// TIA Portal V18 export
FUNCTION "ST10_Main" : Void   // FC1050, LAD
{ S7_Optimized_Access := 'FALSE' }
VERSION : 0.1
// stored: AutoNumber false, IsIECCheckEnabled false, SetENOAutomatically false, UDAEnableTagReadback false
BEGIN

REGION Network 1
   // 系统功能组调用部分
   // 1.该部分用户可以自己根据系统的组成将需要的功能块调用写在该部分
   // 2.该部分禁止与系统功能无关的程序在此处调用
END_REGION

NETWORK
TITLE = XXXX=====Station Relation/工位相关 =====StartXXXXX / XXXX=====Station Relation/Station correlation =====StartXXXXX

REGION Network 3: input /输入
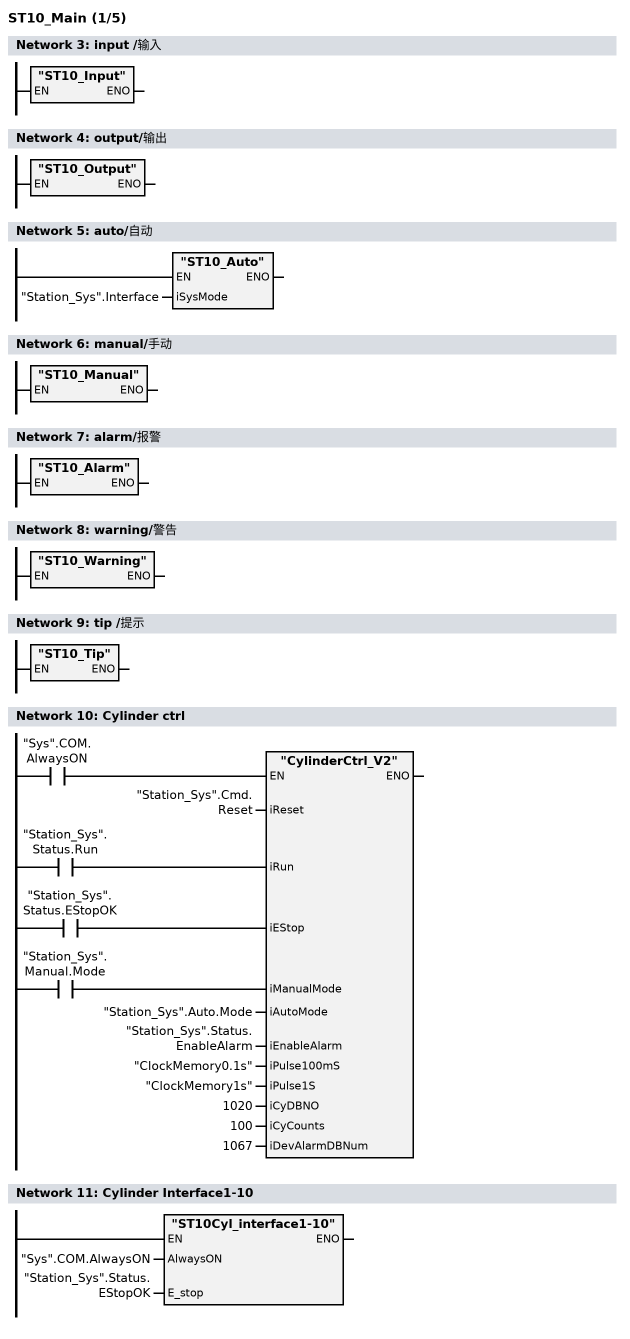
   RUNG wire#powerrail
      "ST10_Input"()
   END_RUNG
   // the same network as SCL:
   "ST10_Input"();
END_REGION

REGION Network 4: output/输出
   RUNG wire#powerrail
      "ST10_Output"()
   END_RUNG
   // the same network as SCL:
   "ST10_Output"();
END_REGION

REGION Network 5: auto/自动
   RUNG wire#powerrail
      "ST10_Auto"(iSysMode := "Station_Sys".Interface)
   END_RUNG
   // the same network as SCL:
   "ST10_Auto"(iSysMode := "Station_Sys".Interface);
END_REGION

REGION Network 6: manual/手动
   RUNG wire#powerrail
      "ST10_Manual"()
   END_RUNG
   // the same network as SCL:
   "ST10_Manual"();
END_REGION

REGION Network 7: alarm/报警
   RUNG wire#powerrail
      "ST10_Alarm"()
   END_RUNG
   // the same network as SCL:
   "ST10_Alarm"();
END_REGION

REGION Network 8: warning/警告
   RUNG wire#powerrail
      "ST10_Warning"()
   END_RUNG
   // the same network as SCL:
   "ST10_Warning"();
END_REGION

REGION Network 9: tip /提示
   RUNG wire#powerrail
      "ST10_Tip"()
   END_RUNG
   // the same network as SCL:
   "ST10_Tip"();
END_REGION

REGION Network 10: Cylinder ctrl
   RUNG wire#powerrail
      Contact( "Sys".COM.AlwaysON )
      "CylinderCtrl_V2"(iRun := wire#w1, iEStop := wire#w2, iManualMode := wire#w3, iReset := "Station_Sys".Cmd.Reset, iAutoMode := "Station_Sys".Auto.Mode, iEnableAlarm := "Station_Sys".Status.EnableAlarm, iPulse100mS := "ClockMemory0.1s", iPulse1S := "ClockMemory1s", iCyDBNO := 1020, iCyCounts := 100, iDevAlarmDBNum := 1067)
   END_RUNG
   RUNG wire#powerrail
      Contact( "Station_Sys".Status.Run )
   END_RUNG wire#w1
   RUNG wire#powerrail
      Contact( "Station_Sys".Status.EStopOK )
   END_RUNG wire#w2
   RUNG wire#powerrail
      Contact( "Station_Sys".Manual.Mode )
   END_RUNG wire#w3
   // the same network as SCL:
   IF "Sys".COM.AlwaysON THEN
       "CylinderCtrl_V2"(iReset := "Station_Sys".Cmd.Reset,
                         iRun := "Station_Sys".Status.Run,
                         iEStop := "Station_Sys".Status.EStopOK,
                         iManualMode := "Station_Sys".Manual.Mode,
                         iAutoMode := "Station_Sys".Auto.Mode,
                         iEnableAlarm := "Station_Sys".Status.EnableAlarm,
                         iPulse100mS := "ClockMemory0.1s",
                         iPulse1S := "ClockMemory1s",
                         iCyDBNO := 1020,
                         iCyCounts := 100,
                         iDevAlarmDBNum := 1067);
   END_IF;
END_REGION

REGION Network 11: Cylinder Interface1-10
   RUNG wire#powerrail
      "ST10Cyl_interface1-10"(AlwaysON := "Sys".COM.AlwaysON, E_stop := "Station_Sys".Status.EStopOK)
   END_RUNG
   // the same network as SCL:
   "ST10Cyl_interface1-10"(AlwaysON := "Sys".COM.AlwaysON, E_stop := "Station_Sys".Status.EStopOK);
END_REGION

REGION Network 12: Cylinder Interface11-20
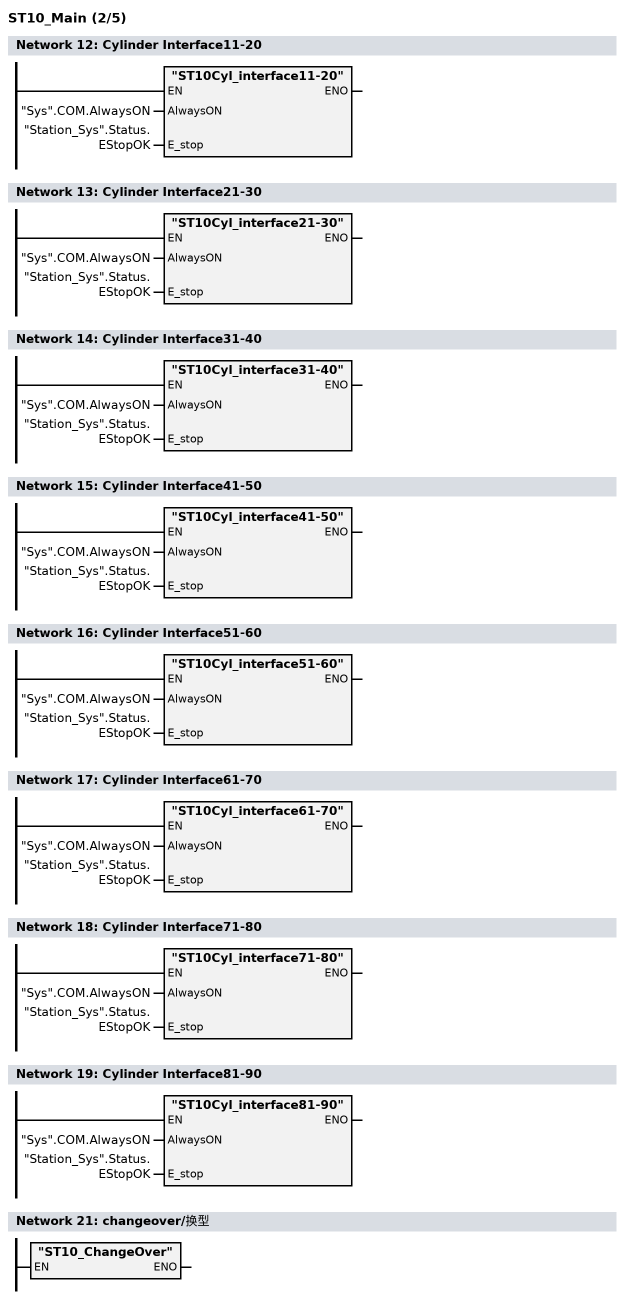
   RUNG wire#powerrail
      "ST10Cyl_interface11-20"(AlwaysON := "Sys".COM.AlwaysON, E_stop := "Station_Sys".Status.EStopOK)
   END_RUNG
   // the same network as SCL:
   "ST10Cyl_interface11-20"(AlwaysON := "Sys".COM.AlwaysON, E_stop := "Station_Sys".Status.EStopOK);
END_REGION

REGION Network 13: Cylinder Interface21-30
   RUNG wire#powerrail
      "ST10Cyl_interface21-30"(AlwaysON := "Sys".COM.AlwaysON, E_stop := "Station_Sys".Status.EStopOK)
   END_RUNG
   // the same network as SCL:
   "ST10Cyl_interface21-30"(AlwaysON := "Sys".COM.AlwaysON, E_stop := "Station_Sys".Status.EStopOK);
END_REGION

REGION Network 14: Cylinder Interface31-40
   RUNG wire#powerrail
      "ST10Cyl_interface31-40"(AlwaysON := "Sys".COM.AlwaysON, E_stop := "Station_Sys".Status.EStopOK)
   END_RUNG
   // the same network as SCL:
   "ST10Cyl_interface31-40"(AlwaysON := "Sys".COM.AlwaysON, E_stop := "Station_Sys".Status.EStopOK);
END_REGION

REGION Network 15: Cylinder Interface41-50
   RUNG wire#powerrail
      "ST10Cyl_interface41-50"(AlwaysON := "Sys".COM.AlwaysON, E_stop := "Station_Sys".Status.EStopOK)
   END_RUNG
   // the same network as SCL:
   "ST10Cyl_interface41-50"(AlwaysON := "Sys".COM.AlwaysON, E_stop := "Station_Sys".Status.EStopOK);
END_REGION

REGION Network 16: Cylinder Interface51-60
   RUNG wire#powerrail
      "ST10Cyl_interface51-60"(AlwaysON := "Sys".COM.AlwaysON, E_stop := "Station_Sys".Status.EStopOK)
   END_RUNG
   // the same network as SCL:
   "ST10Cyl_interface51-60"(AlwaysON := "Sys".COM.AlwaysON, E_stop := "Station_Sys".Status.EStopOK);
END_REGION

REGION Network 17: Cylinder Interface61-70
   RUNG wire#powerrail
      "ST10Cyl_interface61-70"(AlwaysON := "Sys".COM.AlwaysON, E_stop := "Station_Sys".Status.EStopOK)
   END_RUNG
   // the same network as SCL:
   "ST10Cyl_interface61-70"(AlwaysON := "Sys".COM.AlwaysON, E_stop := "Station_Sys".Status.EStopOK);
END_REGION

REGION Network 18: Cylinder Interface71-80
   RUNG wire#powerrail
      "ST10Cyl_interface71-80"(AlwaysON := "Sys".COM.AlwaysON, E_stop := "Station_Sys".Status.EStopOK)
   END_RUNG
   // the same network as SCL:
   "ST10Cyl_interface71-80"(AlwaysON := "Sys".COM.AlwaysON, E_stop := "Station_Sys".Status.EStopOK);
END_REGION

REGION Network 19: Cylinder Interface81-90
   RUNG wire#powerrail
      "ST10Cyl_interface81-90"(AlwaysON := "Sys".COM.AlwaysON, E_stop := "Station_Sys".Status.EStopOK)
   END_RUNG
   // the same network as SCL:
   "ST10Cyl_interface81-90"(AlwaysON := "Sys".COM.AlwaysON, E_stop := "Station_Sys".Status.EStopOK);
END_REGION

REGION Network 21: changeover/换型
   RUNG wire#powerrail
      "ST10_ChangeOver"()
   END_RUNG
   // the same network as SCL:
   "ST10_ChangeOver"();
END_REGION

REGION Network 22: Device
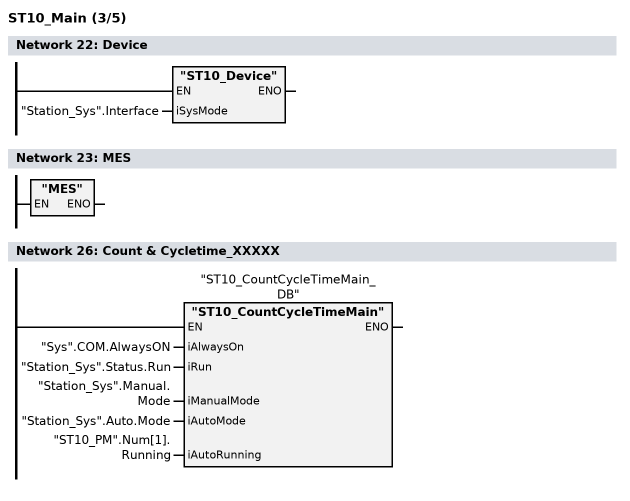
   RUNG wire#powerrail
      "ST10_Device"(iSysMode := "Station_Sys".Interface)
   END_RUNG
   // the same network as SCL:
   "ST10_Device"(iSysMode := "Station_Sys".Interface);
END_REGION

REGION Network 23: MES
   RUNG wire#powerrail
      "MES"()
   END_RUNG
   // the same network as SCL:
   "MES"();
END_REGION

REGION Network 24: =====System Function related information Section =====Start
END_REGION

NETWORK
TITLE = SystemFunction IO

REGION Network 26: Count & Cycletime_XXXXX
   RUNG wire#powerrail
      "ST10_CountCycleTimeMain_DB"(iAlwaysOn := "Sys".COM.AlwaysON, iRun := "Station_Sys".Status.Run, iManualMode := "Station_Sys".Manual.Mode, iAutoMode := "Station_Sys".Auto.Mode, iAutoRunning := "ST10_PM".Num[1].Running)
   END_RUNG
   // the same network as SCL:
   "ST10_CountCycleTimeMain_DB"(iAlwaysOn := "Sys".COM.AlwaysON,   // "ST10_CountCycleTimeMain"
                           iRun := "Station_Sys".Status.Run,
                           iManualMode := "Station_Sys".Manual.Mode,
                           iAutoMode := "Station_Sys".Auto.Mode,
                           iAutoRunning := "ST10_PM".Num[1].Running);
END_REGION

REGION Network 27: System mode
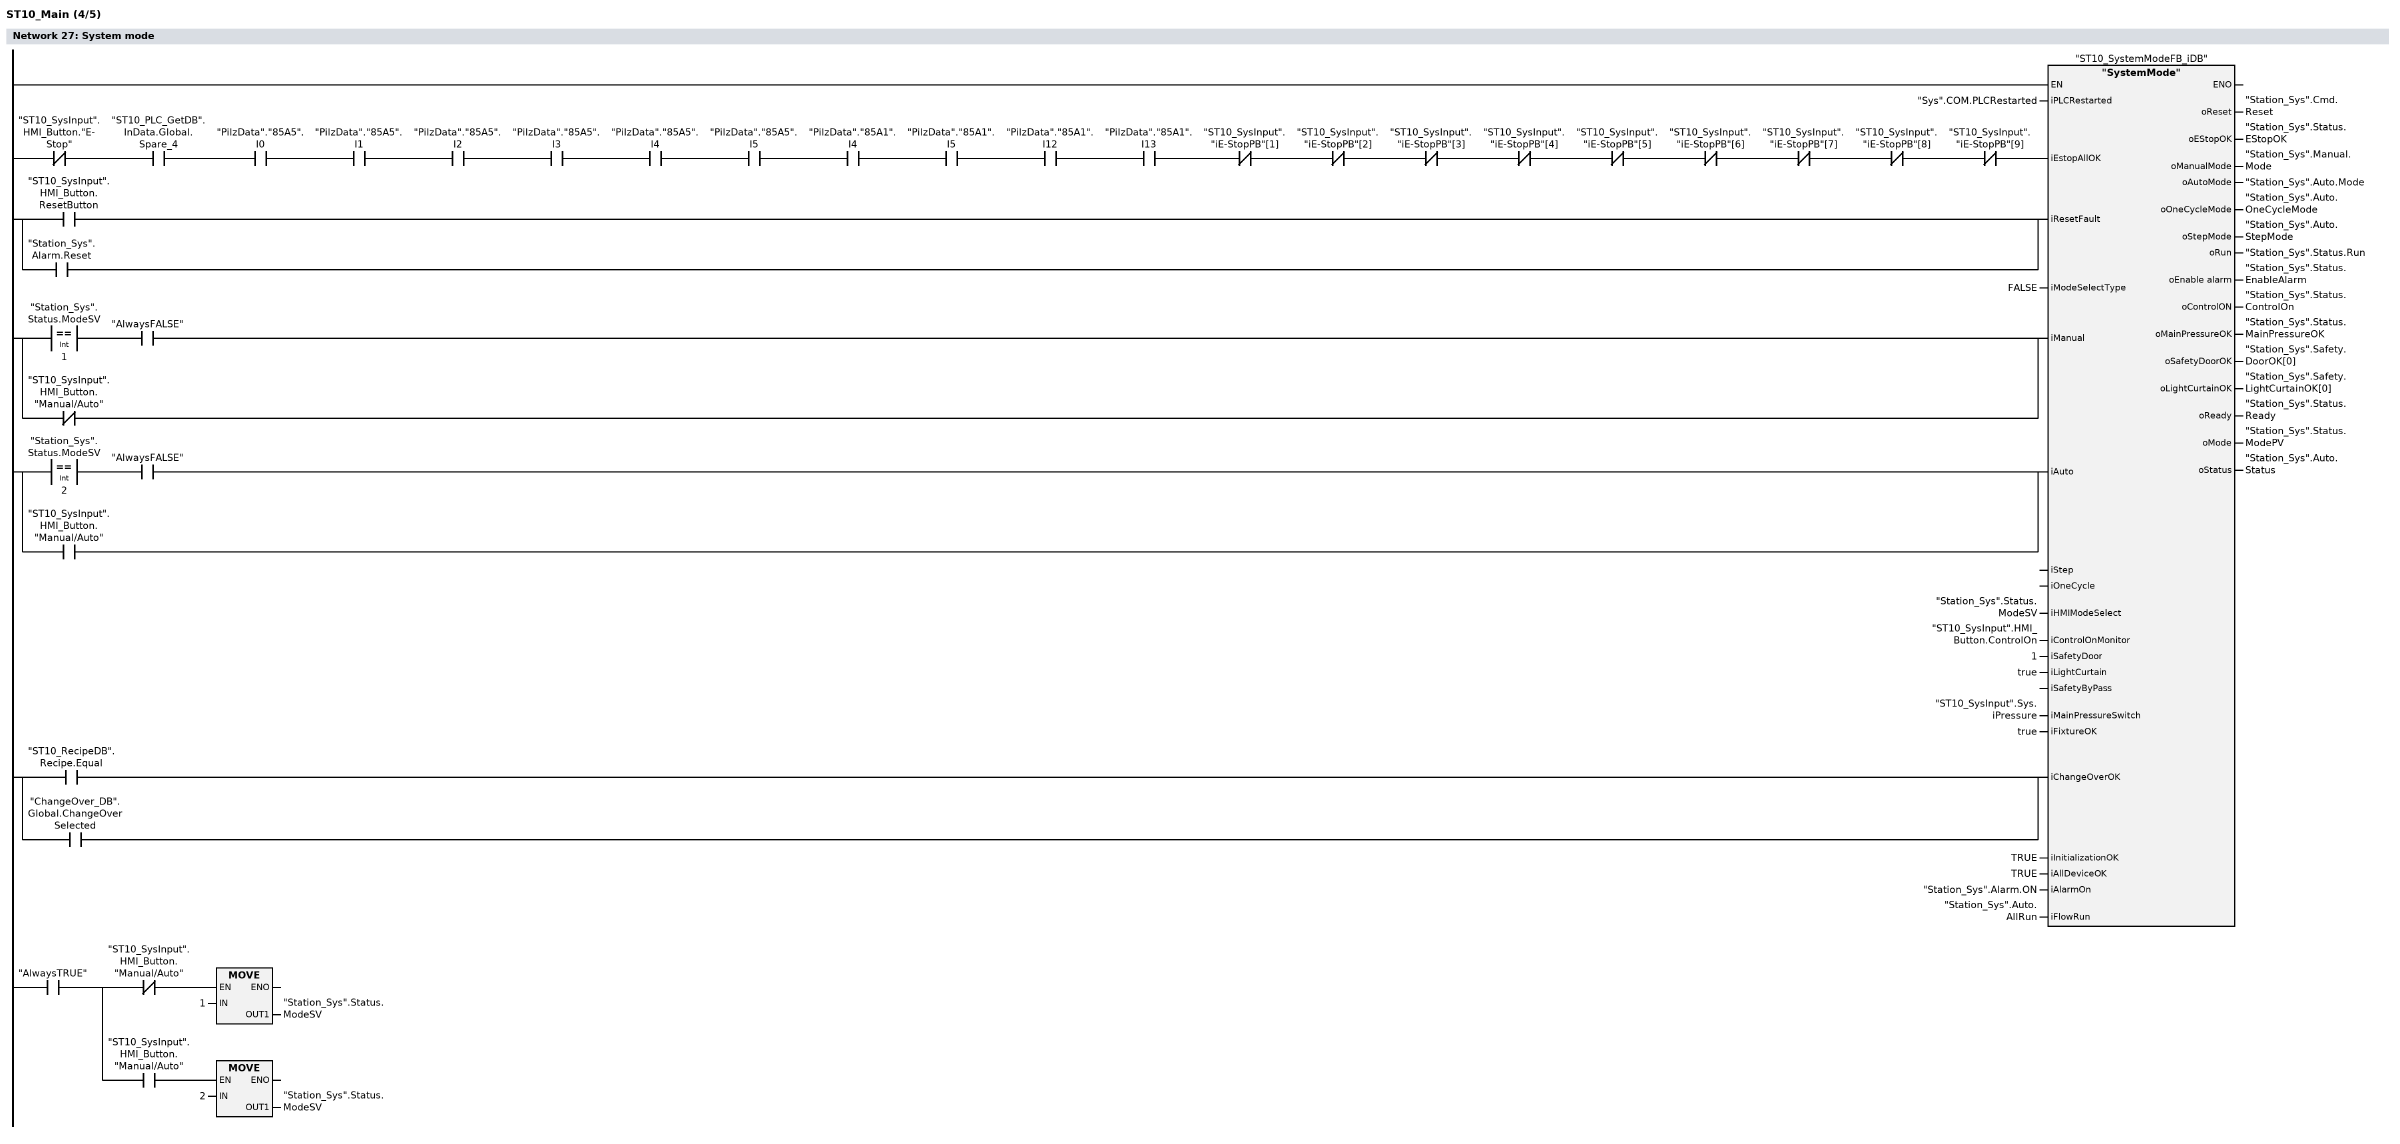
   RUNG wire#powerrail
      "ST10_SystemModeFB_iDB"(iEstopAllOK := wire#w1, iResetFault := wire#w2, iManual := wire#w3, iAuto := wire#w4, iChangeOverOK := wire#w5, iPLCRestarted := "Sys".COM.PLCRestarted, iModeSelectType := FALSE, iStep :=, iOneCycle :=, iHMIModeSelect := "Station_Sys".Status.ModeSV, iControlOnMonitor := "ST10_SysInput".HMI_Button.ControlOn, iSafetyDoor := 1, iLightCurtain := true, iSafetyByPass :=, iMainPressureSwitch := "ST10_SysInput".Sys.iPressure, iFixtureOK := true, iInitializationOK := TRUE, iAllDeviceOK := TRUE, iAlarmOn := "Station_Sys".Alarm.ON, iFlowRun := "Station_Sys".Auto.AllRun, oReset => "Station_Sys".Cmd.Reset, oEStopOK => "Station_Sys".Status.EStopOK, oManualMode => "Station_Sys".Manual.Mode, oAutoMode => "Station_Sys".Auto.Mode, oOneCycleMode => "Station_Sys".Auto.OneCycleMode, oStepMode => "Station_Sys".Auto.StepMode, oRun => "Station_Sys".Status.Run, "oEnable alarm" => "Station_Sys".Status.EnableAlarm, oControlON => "Station_Sys".Status.ControlOn, oMainPressureOK => "Station_Sys".Status.MainPressureOK, oSafetyDoorOK => "Station_Sys".Safety.DoorOK[0], oLightCurtainOK => "Station_Sys".Safety.LightCurtainOK[0], oReady => "Station_Sys".Status.Ready, oMode => "Station_Sys".Status.ModePV, oStatus => "Station_Sys".Auto.Status)
   END_RUNG
   RUNG wire#powerrail
      I_Contact( "ST10_SysInput".HMI_Button."E-Stop" )
      Contact( "ST10_PLC_GetDB".InData.Global.Spare_4 )
      Contact( "PilzData"."85A5".I0 )
      Contact( "PilzData"."85A5".I1 )
      Contact( "PilzData"."85A5".I2 )
      Contact( "PilzData"."85A5".I3 )
      Contact( "PilzData"."85A5".I4 )
      Contact( "PilzData"."85A5".I5 )
      Contact( "PilzData"."85A1".I4 )
      Contact( "PilzData"."85A1".I5 )
      Contact( "PilzData"."85A1".I12 )
      Contact( "PilzData"."85A1".I13 )
      I_Contact( "ST10_SysInput"."iE-StopPB"[1] )
      I_Contact( "ST10_SysInput"."iE-StopPB"[2] )
      I_Contact( "ST10_SysInput"."iE-StopPB"[3] )
      I_Contact( "ST10_SysInput"."iE-StopPB"[4] )
      I_Contact( "ST10_SysInput"."iE-StopPB"[5] )
      I_Contact( "ST10_SysInput"."iE-StopPB"[6] )
      I_Contact( "ST10_SysInput"."iE-StopPB"[7] )
      I_Contact( "ST10_SysInput"."iE-StopPB"[8] )
      I_Contact( "ST10_SysInput"."iE-StopPB"[9] )
   END_RUNG wire#w1
   RUNG wire#powerrail
      Contact( "ST10_SysInput".HMI_Button.ResetButton )
   END_RUNG wire#w2
   RUNG wire#powerrail
      Contact( "Station_Sys".Alarm.Reset )
   END_RUNG wire#w2
   RUNG wire#powerrail
      { S7_Templates := "SrcType := Int" } EQ_Contact(in1 := "Station_Sys".Status.ModeSV, in2 := 1)
      Contact( "AlwaysFALSE" )
   END_RUNG wire#w3
   RUNG wire#powerrail
      I_Contact( "ST10_SysInput".HMI_Button."Manual/Auto" )
   END_RUNG wire#w3
   RUNG wire#powerrail
      { S7_Templates := "SrcType := Int" } EQ_Contact(in1 := "Station_Sys".Status.ModeSV, in2 := 2)
      Contact( "AlwaysFALSE" )
   END_RUNG wire#w4
   RUNG wire#powerrail
      Contact( "ST10_SysInput".HMI_Button."Manual/Auto" )
   END_RUNG wire#w4
   RUNG wire#powerrail
      Contact( "ST10_RecipeDB".Recipe.Equal )
   END_RUNG wire#w5
   RUNG wire#powerrail
      Contact( "ChangeOver_DB".Global.ChangeOverSelected )
   END_RUNG wire#w5
   RUNG wire#powerrail
      Contact( "AlwaysTRUE" )
      wire#w6
      I_Contact( "ST10_SysInput".HMI_Button."Manual/Auto" )
      Move(in := 1, out1 => "Station_Sys".Status.ModeSV)
   END_RUNG
   RUNG wire#w6
      Contact( "ST10_SysInput".HMI_Button."Manual/Auto" )
      Move(in := 2, out1 => "Station_Sys".Status.ModeSV)
   END_RUNG
   // the same network as SCL:
   "ST10_SystemModeFB_iDB"(iPLCRestarted := "Sys".COM.PLCRestarted,   // "SystemMode"
                           iEstopAllOK := NOT "ST10_SysInput".HMI_Button."E-Stop" AND "ST10_PLC_GetDB".InData.Global.Spare_4 AND "PilzData"."85A5".I0 AND "PilzData"."85A5".I1 AND "PilzData"."85A5".I2 AND "PilzData"."85A5".I3 AND "PilzData"."85A5".I4 AND "PilzData"."85A5".I5 AND "PilzData"."85A1".I4 AND "PilzData"."85A1".I5 AND "PilzData"."85A1".I12 AND "PilzData"."85A1".I13 AND NOT "ST10_SysInput"."iE-StopPB"[1] AND NOT "ST10_SysInput"."iE-StopPB"[2] AND NOT "ST10_SysInput"."iE-StopPB"[3] AND NOT "ST10_SysInput"."iE-StopPB"[4] AND NOT "ST10_SysInput"."iE-StopPB"[5] AND NOT "ST10_SysInput"."iE-StopPB"[6] AND NOT "ST10_SysInput"."iE-StopPB"[7] AND NOT "ST10_SysInput"."iE-StopPB"[8] AND NOT "ST10_SysInput"."iE-StopPB"[9],
                           iResetFault := "ST10_SysInput".HMI_Button.ResetButton OR "Station_Sys".Alarm.Reset,
                           iModeSelectType := FALSE,
                           iManual := (("Station_Sys".Status.ModeSV = 1) AND "AlwaysFALSE") OR NOT "ST10_SysInput".HMI_Button."Manual/Auto",
                           iAuto := (("Station_Sys".Status.ModeSV = 2) AND "AlwaysFALSE") OR "ST10_SysInput".HMI_Button."Manual/Auto",
                           iHMIModeSelect := "Station_Sys".Status.ModeSV,
                           iControlOnMonitor := "ST10_SysInput".HMI_Button.ControlOn,
                           iSafetyDoor := 1,
                           iLightCurtain := true,
                           iMainPressureSwitch := "ST10_SysInput".Sys.iPressure,
                           iFixtureOK := true,
                           iChangeOverOK := "ST10_RecipeDB".Recipe.Equal OR "ChangeOver_DB".Global.ChangeOverSelected,
                           iInitializationOK := TRUE,
                           iAllDeviceOK := TRUE,
                           iAlarmOn := "Station_Sys".Alarm.ON,
                           iFlowRun := "Station_Sys".Auto.AllRun,
                           oReset => "Station_Sys".Cmd.Reset,
                           oEStopOK => "Station_Sys".Status.EStopOK,
                           oManualMode => "Station_Sys".Manual.Mode,
                           oAutoMode => "Station_Sys".Auto.Mode,
                           oOneCycleMode => "Station_Sys".Auto.OneCycleMode,
                           oStepMode => "Station_Sys".Auto.StepMode,
                           oRun => "Station_Sys".Status.Run,
                           "oEnable alarm" => "Station_Sys".Status.EnableAlarm,
                           oControlON => "Station_Sys".Status.ControlOn,
                           oMainPressureOK => "Station_Sys".Status.MainPressureOK,
                           oSafetyDoorOK => "Station_Sys".Safety.DoorOK[0],
                           oLightCurtainOK => "Station_Sys".Safety.LightCurtainOK[0],
                           oReady => "Station_Sys".Status.Ready,
                           oMode => "Station_Sys".Status.ModePV,
                           oStatus => "Station_Sys".Auto.Status);
   IF "AlwaysTRUE" AND NOT "ST10_SysInput".HMI_Button."Manual/Auto" THEN
       "Station_Sys".Status.ModeSV := 1;
   END_IF;
   IF "AlwaysTRUE" AND "ST10_SysInput".HMI_Button."Manual/Auto" THEN
       "Station_Sys".Status.ModeSV := 2;
   END_IF;
END_REGION

REGION Network 28: Start button
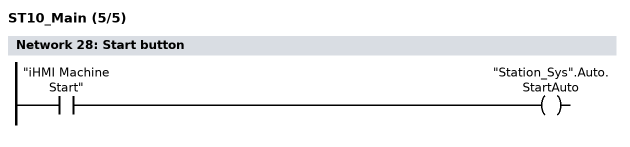
   RUNG wire#powerrail
      Contact( "iHMI Machine Start" )
      Coil( "Station_Sys".Auto.StartAuto )
   END_RUNG
   // the same network as SCL:
   "Station_Sys".Auto.StartAuto := "iHMI Machine Start";
END_REGION

REGION Network 29 (SCL): System Interface
   "Station_Sys".Interface.CPUFristCycle  := "Sys".COM.PLCRestarted;
   "Station_Sys".Interface.SysRun         := "Station_Sys".Status.Run;
   "Station_Sys".Interface.Reset          := "Station_Sys".Cmd.Reset;
   "Station_Sys".Interface.EstopOK        := "Station_Sys".Status.EStopOK;
   "Station_Sys".Interface.SafetyDoorOK   := "Station_Sys".Safety.DoorOK[0];
   "Station_Sys".Interface.LightCurtainOK := "Station_Sys".Safety.LightCurtainOK[0];
   "Station_Sys".Interface.SetInitial     := "Station_Sys".Initial.Set;
   "Station_Sys".Interface.InitialRun     := "Station_Sys".Initial.Running;
   "Station_Sys".Interface.Ready          := "Station_Sys".Status.Ready;
   "Station_Sys".Interface.ManualMode     := "Station_Sys".Manual.Mode;
   "Station_Sys".Interface.Auto           := "Station_Sys".Auto;
END_REGION

REGION Network 30: =====System Function related information Section =====End
END_REGION

REGION Network 31: CallCalibration//标定调用
END_REGION

REGION Network 32 (SCL): ByPass Button
   // A
   "ST10_GeneralData".FunctionDeSelect.A.FunctionDeSelected_Servo380A1  := "ST10_GeneralData".FunctionDeSelect.A.DeSelectPB_Servo380A1;
   "ST10_GeneralData".FunctionDeSelect.A.FunctionDeSelected_Servo381A1  := "ST10_GeneralData".FunctionDeSelect.A.DeSelectPB_Servo381A1;
   "ST10_GeneralData".FunctionDeSelect.A.FunctionDeSelected_Servo383A1  := "ST10_GeneralData".FunctionDeSelect.A.DeSelectPB_Servo383A1;
   "ST10_GeneralData".FunctionDeSelect.A.FunctionDeSelected_Reader800A1 := "ST10_GeneralData".FunctionDeSelect.A.DeSelectPB_Reader800A1;
   "ST10_GeneralData".FunctionDeSelect.A.FunctionDeSelected_Reader801A1 := "ST10_GeneralData".FunctionDeSelect.A.DeSelectPB_Reader801A1;
   "ST10_GeneralData".FunctionDeSelect.A.FunctionDeSelected_Reader802A1 := "ST10_GeneralData".FunctionDeSelect.A.DeSelectPB_Reader802A1;
   "ST10_GeneralData".FunctionDeSelect.A.FunctionDeSelected_Reader803A1 := "ST10_GeneralData".FunctionDeSelect.A.DeSelectPB_Reader803A1;
   "ST10_GeneralData".FunctionDeSelect.A.FunctionDeSelected_Reader804A1 := "ST10_GeneralData".FunctionDeSelect.A.DeSelectPB_Reader804A1;

   // B
   "ST10_GeneralData".FunctionDeSelect.B.FunctionDeSelected_Press372A1     := "ST10_GeneralData".FunctionDeSelect.B.DeSelectPB_Press372A1;
   "ST10_GeneralData".FunctionDeSelect.B.FunctionDeSelected_Press375A1     := "ST10_GeneralData".FunctionDeSelect.B.DeSelectPB_Press375A1;
   "ST10_GeneralData".FunctionDeSelect.B.FunctionDeSelected_Reader806A1    := "ST10_GeneralData".FunctionDeSelect.B.DeSelectPB_Reader806A1;
   "ST10_GeneralData".FunctionDeSelect.B.FunctionDeSelected_TestPress372A1 := "ST10_GeneralData".FunctionDeSelect.B.DeSelectPB_TestPress372A1;
   "ST10_GeneralData".FunctionDeSelect.B.FunctionDeSelected_TestPress375A1 := "ST10_GeneralData".FunctionDeSelect.B.DeSelectPB_TestPress375A1;

   // C
   "ST10_GeneralData".FunctionDeSelect.C.FunctionDeSelected_Servo382A1 := "ST10_GeneralData".FunctionDeSelect.C.DeSelectPB_Servo382A1;
   "ST10_GeneralData".FunctionDeSelect.C.FunctionDeSelected_ServoIAI := "ST10_GeneralData".FunctionDeSelect.C.DeSelectPB_ServoIAI;
   "ST10_GeneralData".FunctionDeSelect.C.FunctionDeSelected_IV3810A1 := "ST10_GeneralData".FunctionDeSelect.C.DeSelectPB_IV3810A1;
   "ST10_GeneralData".FunctionDeSelect.C.FunctionDeSelected_IV3811A1 := "ST10_GeneralData".FunctionDeSelect.C.DeSelectPB_IV3811A1;
   "ST10_GeneralData".FunctionDeSelect.C.FunctionDeSelected_Glue := "ST10_GeneralData".FunctionDeSelect.C.DeSelectPB_Glue;

   // E
   "ST10_GeneralData".FunctionDeSelect.E.FunctionDeSelected := "ST10_GeneralData".FunctionDeSelect.E.DeSelectPB;

   // F
   "ST10_GeneralData".FunctionDeSelect.F.FunctionDeSelected_Reader805A1 := "ST10_GeneralData".FunctionDeSelect.F.DeSelectPB_Reader805A1;

   // H
   "ST10_GeneralData".FunctionDeSelect.H.FunctionDeSelected := "ST10_GeneralData".FunctionDeSelect.H.DeSelectPB;

   // J
   "ST10_GeneralData".FunctionDeSelect.J.FunctionDeSelected := "ST10_GeneralData".FunctionDeSelect.J.DeSelectPB;

   // K
   "ST10_GeneralData".FunctionDeSelect.K.FunctionDeSelected := "ST10_GeneralData".FunctionDeSelect.K.DeSelectPB;

   // L
   "ST10_GeneralData".FunctionDeSelect.L.FunctionDeSelected := "ST10_GeneralData".FunctionDeSelect.L.DeSelectPB;

   // MES
   "ST10_GeneralData".FunctionDeSelect.MES.FunctionDeSelected := "ST10_GeneralData".FunctionDeSelect.MES.DeSelectPB;

   //Auto>Maanual  ScanFixture
   "ST10_GeneralData".FunctionDeSelect.Global.FunctionDeSelected_ScanFixture := "ST10_GeneralData".FunctionDeSelect.Global.DeSelectPB_ScanFixture;
END_REGION
END_FUNCTION
